(* IEC 61131-3 sources: Laboratorijsko-busace-postrojenje/Libraries/dvframe, 3 files *)

(* ---- dvframe.typ ---- *)
(********************************************************************
 * COPYRIGHT (C) BERNECKER + RAINER, AUSTRIA, A-5142 EGGELSBERG
 ********************************************************************
 * Library: DVFrame
 * File: DVFrame.typ
 * Created: 11.11.2003
 ********************************************************************
 * Global data types of library DVFrame
 ********************************************************************)
TYPE
	XOPENCONFIG : STRUCT
		idle	: UINT ;					(*maximum idle time between characters*)
		delimc	: UINT ;					(*activate the frame delimiters, standard value : 0*)
		delim	: ARRAY[0..1] OF USINT ;	(*frame delimiters, default value: 0,0*)
		tx_cnt	: UINT ;					(*number of send buffers (maximum 8), default value: 2*)
		rx_cnt	: UINT ;					(*number of receive buffers (maximum 8), default value: 2*)
		tx_len	: UINT ;					(*send buffer length, default value: 256 bytes*)
		rx_len	: UINT ;					(*receive buffer length, default value: 256 bytes*)
		argc	: UINT ;					(*number of additional arguments in argv, default value: 0*)
		argv	: UDINT ;					(*address for a UDINT field with additional arguments, default value: 0*)
	END_STRUCT;
END_TYPE

(* ---- dvframe.fun ---- *)
(********************************************************************
 * COPYRIGHT (C) BERNECKER + RAINER, AUSTRIA, A-5142 EGGELSBERG
 ********************************************************************
 * Library: DVFrame
 * File: DVFrame.fun
 * Created: 11.11.2003
 ********************************************************************
 * Functions and function blocks of library DVFrame
 ********************************************************************)
FUNCTION_BLOCK FRM_mode				(*modifies the values for the baud rate and asynchronous parameters*)
	VAR_INPUT
		enable	:BOOL;				(*enables execution*)
		ident	:UDINT;				(*driver ID for the interface (see FRM_xopen())*)
		mode	:UDINT;				(*address of the string which configures the interface to be used*)
	END_VAR
	VAR_OUTPUT
		status	:UINT;				(*execution status: ERR_OK, ERR_FUB_ENABLE_FALSE, 0xXXXX = see help*)
	END_VAR
	VAR
		internal	:STRING[27];	(*internal variable*)
	END_VAR
END_FUNCTION_BLOCK

FUNCTION_BLOCK FRM_ctrl				(*operates the DSR/DTR signals for modem capable interfaces*)
	VAR_INPUT
		enable	:BOOL;				(*enables execution*)
		ident	:UDINT;				(*driver ID for the interface (see FRM_xopen())*)
		ioctrl	:UINT;				(*control selection*)
		inarg	:UDINT;				(*input argument*)
	END_VAR
	VAR_OUTPUT
		status	:UINT;				(*execution status: ERR_OK, ERR_FUB_ENABLE_FALSE, 0xXXXX = see help*)
		outarg	:UDINT;				(*output argument*)
	END_VAR
	VAR
		internal	:STRING[43];	(*internal variable*)
	END_VAR
END_FUNCTION_BLOCK

FUNCTION_BLOCK FRM_robuf			(*releases the send buffer manually*)
	VAR_INPUT
		enable	:BOOL;				(*enables execution*)
		ident	:UDINT;				(*driver ID for the interface (see FRM_xopen())*)
		buffer	:UDINT;				(*send buffer address*)
		buflng	:UINT;				(*send buffer length*)
	END_VAR
	VAR_OUTPUT
		status	:UINT;				(*execution status: ERR_OK, ERR_FUB_ENABLE_FALSE, 0xXXXX = see help*)
	END_VAR
	VAR
		internal	:STRING[27];	(*internal variable*)
	END_VAR
END_FUNCTION_BLOCK

FUNCTION_BLOCK FRM_gbuf				(*requests an available send buffer*)
	VAR_INPUT
		enable	:BOOL;				(*enables execution*)
		ident	:UDINT;				(*driver ID for the interface (see FRM_xopen())*)
	END_VAR
	VAR_OUTPUT
		status	:UINT;				(*execution status: ERR_OK, ERR_FUB_ENABLE_FALSE, 0xXXXX = see help*)
		buffer	:UDINT;				(*send buffer address*)
		buflng	:UINT;				(*send buffer length*)
	END_VAR
	VAR
		internal	:STRING[27];	(*internal variable*)
	END_VAR
END_FUNCTION_BLOCK

FUNCTION_BLOCK FRM_rbuf				(*releases the receive buffer*)
	VAR_INPUT
		enable	:BOOL;				(*enables execution*)
		ident	:UDINT;				(*driver ID for the interface (see FRM_xopen())*)
		buffer	:UDINT;				(*receive buffer address*)
		buflng	:UINT;				(*receive buffer length*)
	END_VAR
	VAR_OUTPUT
		status	:UINT;				(*execution status: ERR_OK, ERR_FUB_ENABLE_FALSE, 0xXXXX = see help*)
	END_VAR
	VAR
		internal	:STRING[27];	(*internal variable*)
	END_VAR
END_FUNCTION_BLOCK

FUNCTION_BLOCK FRM_close			(*uses the DVFRAME.BR (or DVFRAME3.BR) frame driver*)
	VAR_INPUT
		enable	:BOOL;				(*enables execution*)
		ident	:UDINT;				(*driver ID for the interface (see FRM_xopen())*)
	END_VAR
	VAR_OUTPUT
		status	:UINT;				(*execution status: ERR_OK, ERR_FUB_ENABLE_FALSE, 0xXXXX = see help*)
	END_VAR
	VAR
		internal	:STRING[27];	(*internal variable*)
	END_VAR
END_FUNCTION_BLOCK

FUNCTION_BLOCK FRM_write			(*enables the frame driver to send data to the send buffer*)
	VAR_INPUT
		enable	:BOOL;				(*enables execution*)
		ident	:UDINT;				(*driver ID for the interface (see FRM_xopen())*)
		buffer	:UDINT;				(*send buffer address*)
		buflng	:UINT;				(*send buffer length*)
	END_VAR
	VAR_OUTPUT
		status	:UINT;				(*execution status: ERR_OK, ERR_FUB_ENABLE_FALSE, 0xXXXX = see help*)
	END_VAR
	VAR
		internal	:STRING[27];	(*internal variable*)
	END_VAR
END_FUNCTION_BLOCK

FUNCTION_BLOCK FRM_read				(*starts the receive process*)
	VAR_INPUT
		enable	:BOOL;				(*enables execution*)
		ident	:UDINT;				(*driver ID for the interface (see FRM_xopen())*)
	END_VAR
	VAR_OUTPUT
		status	:UINT;				(*execution status: ERR_OK, ERR_FUB_ENABLE_FALSE, 0xXXXX = see help*)
		buffer	:UDINT;				(*receive buffer address*)
		buflng	:UINT;				(*receive buffer length*)
	END_VAR
	VAR
		internal	:STRING[27];	(*internal variable*)
	END_VAR
END_FUNCTION_BLOCK

FUNCTION_BLOCK FRM_xopen			(*initializes and prepares up to 16 interfaces for frame transfer*)
	VAR_INPUT
		enable	:BOOL;				(*enables execution*)
		device	:UDINT;				(*pointer to a string which clearly describes the interface used*)
		mode	:UDINT;				(*pointer to the string which configures the interface to be used*)
		config	:UDINT;				(*address for a configuration structure can be entered at this point (optional entry)*)
	END_VAR
	VAR_OUTPUT
		status	:UINT;				(*execution status: ERR_OK, ERR_FUB_ENABLE_FALSE, 0xXXXX = see help*)
		ident	:UDINT;				(*driver ID for the interface (required for other functions in the DVFrame library)*)
	END_VAR
	VAR
		internal	:STRING[27];	(*internal variable*)
	END_VAR
END_FUNCTION_BLOCK

(* ---- dvframe.var ---- *)
(********************************************************************
 * COPYRIGHT (C) BERNECKER + RAINER, AUSTRIA, A-5142 EGGELSBERG
 ********************************************************************
 * Library:    DVFrame
 * File:            DVFrame.var
 * Created:         11.11.2003
 ********************************************************************
 * Constants of library DVFrame
 ********************************************************************)
VAR CONSTANT
	frmERR_IOCTL_NOTSUPPORTED	: UINT	:= 8257;	(*command not supported by driver (hardware)*)
	frmERR_DEVICEDESCRIPTION	: UINT	:= 8252;	(*device not found*)
	frmERR_FUB_ENABLE_FALSE	: UINT	:= 65534;
	frmERR_TRANSMITOVERRUN	: UINT	:= 8078;		(*send buffer waiting queue full*)
	frmERR_MODEDESCRIPTION	: UINT	:= 8253;		(*syntax error in mode parameter string, or mode parameter not supported by the specified device*)
	frmERR_IOCTL_NOTVALID	: UINT	:= 8073;		(*invalid I/O control code*)
	frmERR_INVALIDBUFFER	: UINT	:= 8072;		(*invalid buffer rejected*)
	ARG_EVSEND_TASKIDENT	: UDINT	:= 14;
	ARG_EVSEND_TASKEVENT	: UDINT	:= 18;
	frmERR_NORESOURCES	: UINT	:= 8258;			(*required resource not available (memory, OS object, etc.)*)
	frmERR_INPUTERROR	: UINT	:= 8079;			(*frame buffer with defective character*)
	frmERR_NOTOPENED	: UINT	:= 8251;			(*device not open*)
	MISC_RECEIVE_ALL	: UDINT	:= 2;
	frmERR_PA_DB_SB	: UINT	:= 8256;				(*/PA, /DB, /SB must always be specified together*)
	frmERR_NOBUFFER	: UINT	:= 8071;				(*no buffer available in the send buffer manager*)
	ARG_TXPVPOLLADR	: UDINT	:= 17;
	frmERR_NOINPUT	: UINT	:= 60;					(*no message received*)
	frmERR_MAXOPEN	: UINT	:= 8254;				(*too many devices opened at once*)
	ARG_PVPOLLADR	: UDINT	:= 15;
	frmERR_OK	: UINT	:= 0;
	ARG_MISC	: UDINT	:= 16;
	ARG_BAUD	: UDINT	:= 0;
END_VAR
